ORGANIZATION_BLOCK MAIN:OB1
TITLE=PROGRAM COMMENTS
BEGIN
Network 1 // Network Title
// Network Comment
LD     I0.1
A      I0.2
A      I0.3
=      Q0.0
Network 2
LDN    I0.1
A      I0.3
LDN    I0.2
A      I0.3
OLD
LD     I0.1
A      I0.2
AN     I0.3
OLD
=      Q0.1
Network 3
LDN    I0.1
A      I0.2
LD     I0.1
AN     I0.2
OLD
=      Q0.2
Network 4
LD     I0.0
=      Q0.3
END_ORGANIZATION_BLOCK
SUBROUTINE_BLOCK SBR_0:SBR0
TITLE=SUBROUTINE COMMENTS
BEGIN
Network 1 // Network Title
// Network Comment
END_SUBROUTINE_BLOCK
INTERRUPT_BLOCK INT_0:INT0
TITLE=INTERRUPT ROUTINE COMMENTS
BEGIN
Network 1 // Network Title
// Network Comment
END_INTERRUPT_BLOCK
